Staubli VAL3: JointPos.dtx

public jointRx JointPos
